Omron CX-Programmer project NewProject (CX-Programmer 9.75)

# PLC PLCGROUP4: CPM2* 

## Global symbols (name address type ; comment)
0.00 BOOL  ; GO_Default
0.01 BOOL  ; IN_PB_1
0.02 BOOL  ; IN_PB_2
0.03 BOOL  ; IN_PB_3
0.04 BOOL  ; SF_FLOOR_1
0.05 BOOL  ; SF_FLOOR_2
0.06 BOOL  ; SF_FLOOR_3
0.07 BOOL  ; SD_CAGE_LIMIT_OPEN
0.08 BOOL  ; SD_CAGE_LIMIT_CLOSE
0.09 BOOL  ; S1_OPEN
0.10 BOOL  ; S1_CLOSE
0.11 BOOL  ; SF_FLOOR_1
0.12 BOOL  ; SF_FLOOR_2
0.13 BOOL  ; SF_FLOOR_3
0.14 BOOL  ; CD_CAGE_LIMIT_OPEN
0.15 BOOL  ; SD_CAGE_LIMIT_CLOSE
10.00 BOOL  ; MOTOR_UP
10.01 BOOL  ; MOTOR_DOWN
10.02 BOOL  ; OPEN_CABIN
10.03 BOOL  ; CLOSE_CABIN
10.04 BOOL  ; M1_OPEN
10.05 BOOL  ; M1_CLOSE
10.06 BOOL  ; M2_OPEN
10.07 BOOL  ; M2_CLOSE
11.00 BOOL  ; M3_OPEN
11.01 BOOL  ; M3_CLOSE
1.00 BOOL  ; S2_OPEN
1.01 BOOL  ; S2_CLOSED
1.02 BOOL  ; S3_OPEN
1.03 BOOL  ; S3_CLOSED
1.04 BOOL  ; SD_CAGE_LIMIT_OPEN
1.05 BOOL  ; SD_CAGE_LIMIT_CLOSE
9.00 BOOL  ; GO_FLOOR_1
9.01 BOOL  ; GO_FLOOR_2
9.02 BOOL  ; GO_FLOOR_3
9.03 BOOL  ; GO_DOWN_FLAG
9.04 BOOL  ; GO_UP_FLAG
9.05 BOOL  ; OPEN_CABIN/FLOOR_DOOR
9.06 BOOL  ; OPEN_DOOR_F1
9.07 BOOL  ; OPEN_DOOR_F2
9.08 BOOL  ; OPEN_DOOR_F3
9.09 BOOL  ; DONE_1
9.10 BOOL  ; DONE_2
9.11 BOOL  ; DONE_3
TIM000 BOOL  ; TIMER CABIN
TIM001 BOOL  ; TIMER_FLOOR_1_DOOR
TIM002 BOOL  ; TIMER_FLOOR_2_DOOR
TIM004 BOOL  ; \

## Program NewProgram1 (no task)
; Lift Code
Local symbols
SF_FLOOR_3 BOOL

### Section Test_Code

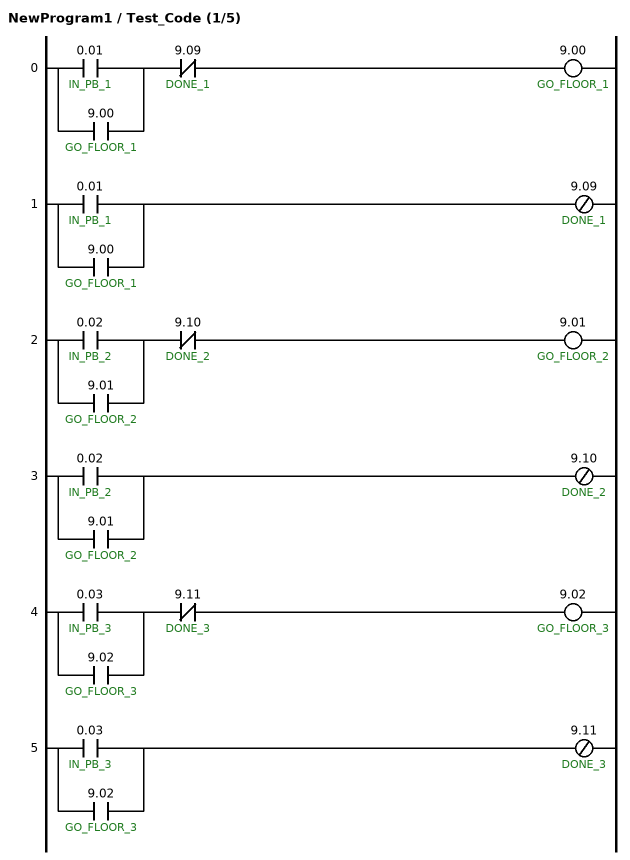
; rung 0
LD 0.01  ; IN_PB_1
OR 9.00  ; GO_FLOOR_1
ANDNOT 9.09  ; DONE_1
OUT 9.00  ; GO_FLOOR_1
; rung 1
LD 0.01  ; IN_PB_1
OR 9.00  ; GO_FLOOR_1
OUTNOT 9.09  ; DONE_1
; rung 2
LD 0.02  ; IN_PB_2
OR 9.01  ; GO_FLOOR_2
ANDNOT 9.10  ; DONE_2
OUT 9.01  ; GO_FLOOR_2
; rung 3
LD 0.02  ; IN_PB_2
OR 9.01  ; GO_FLOOR_2
OUTNOT 9.10  ; DONE_2
; rung 4
LD 0.03  ; IN_PB_3
OR 9.02  ; GO_FLOOR_3
ANDNOT 9.11  ; DONE_3
OUT 9.02  ; GO_FLOOR_3
; rung 5
LD 0.03  ; IN_PB_3
OR 9.02  ; GO_FLOOR_3
OUTNOT 9.11  ; DONE_3

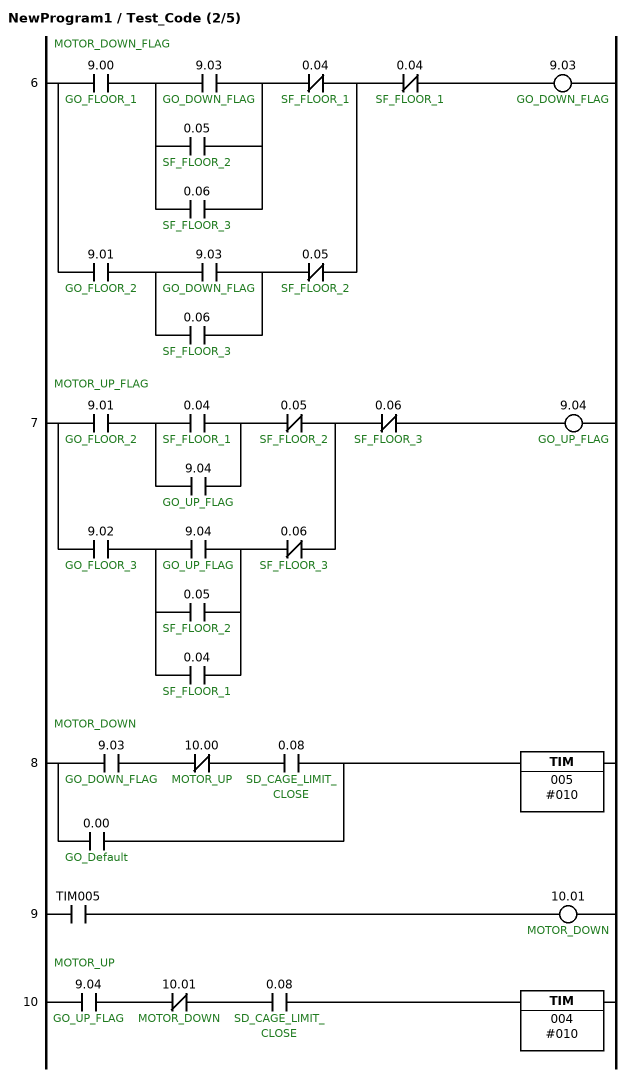
; rung 6: MOTOR_DOWN_FLAG
LD 9.00  ; GO_FLOOR_1
LD 9.03  ; GO_DOWN_FLAG
OR 0.05  ; SF_FLOOR_2
OR 0.06  ; SF_FLOOR_3
ANDLD
ANDNOT 0.04  ; SF_FLOOR_1
LD 9.01  ; GO_FLOOR_2
LD 9.03  ; GO_DOWN_FLAG
OR 0.06  ; SF_FLOOR_3
ANDLD
ANDNOT 0.05  ; SF_FLOOR_2
ORLD
ANDNOT 0.04  ; SF_FLOOR_1
OUT 9.03  ; GO_DOWN_FLAG
; rung 7: MOTOR_UP_FLAG
LD 9.01  ; GO_FLOOR_2
LD 0.04  ; SF_FLOOR_1
OR 9.04  ; GO_UP_FLAG
ANDLD
ANDNOT 0.05  ; SF_FLOOR_2
LD 9.02  ; GO_FLOOR_3
LD 9.04  ; GO_UP_FLAG
OR 0.05  ; SF_FLOOR_2
OR 0.04  ; SF_FLOOR_1
ANDLD
ANDNOT 0.06  ; SF_FLOOR_3
ORLD
ANDNOT 0.06  ; SF_FLOOR_3
OUT 9.04  ; GO_UP_FLAG
; rung 8: MOTOR_DOWN
LD 9.03  ; GO_DOWN_FLAG
ANDNOT 10.00  ; MOTOR_UP
AND 0.08  ; SD_CAGE_LIMIT_CLOSE
OR 0.00  ; GO_Default
TIM 005 #010
; rung 9
LD TIM005
OUT 10.01  ; MOTOR_DOWN
; rung 10: MOTOR_UP
LD 9.04  ; GO_UP_FLAG
ANDNOT 10.01  ; MOTOR_DOWN
AND 0.08  ; SD_CAGE_LIMIT_CLOSE
TIM 004 #010

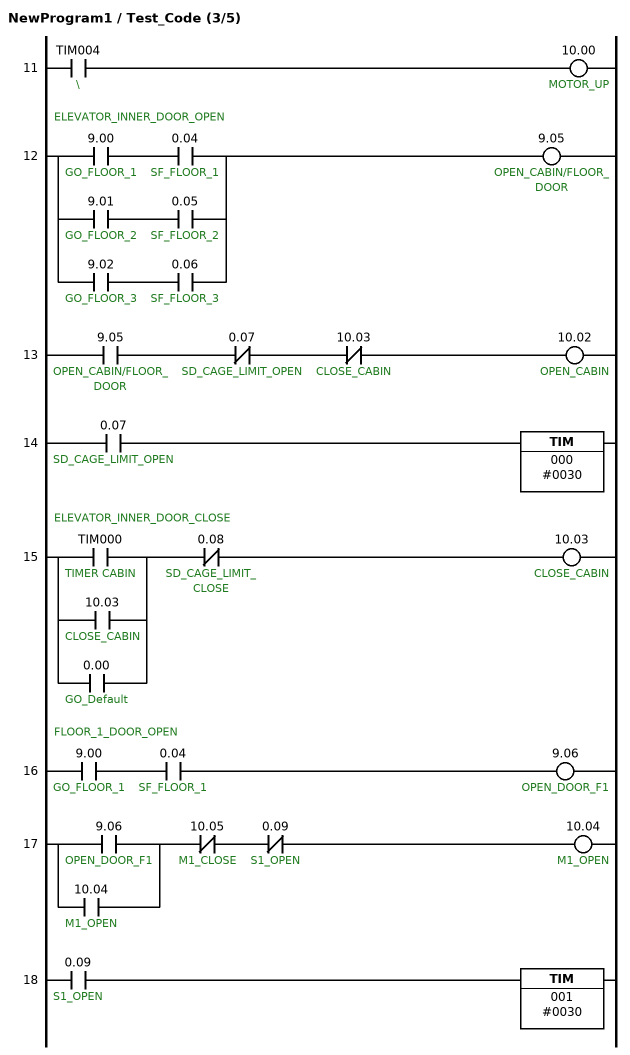
; rung 11
LD TIM004  ; \
OUT 10.00  ; MOTOR_UP
; rung 12: ELEVATOR_INNER_DOOR_OPEN
LD 9.00  ; GO_FLOOR_1
AND 0.04  ; SF_FLOOR_1
LD 9.01  ; GO_FLOOR_2
AND 0.05  ; SF_FLOOR_2
ORLD
LD 9.02  ; GO_FLOOR_3
AND 0.06  ; SF_FLOOR_3
ORLD
OUT 9.05  ; OPEN_CABIN/FLOOR_DOOR
; rung 13
LD 9.05  ; OPEN_CABIN/FLOOR_DOOR
ANDNOT 0.07  ; SD_CAGE_LIMIT_OPEN
ANDNOT 10.03  ; CLOSE_CABIN
OUT 10.02  ; OPEN_CABIN
; rung 14
LD 0.07  ; SD_CAGE_LIMIT_OPEN
TIM 000 #0030
; rung 15: ELEVATOR_INNER_DOOR_CLOSE
LD TIM000  ; TIMER CABIN
OR 10.03  ; CLOSE_CABIN
OR 0.00  ; GO_Default
ANDNOT 0.08  ; SD_CAGE_LIMIT_CLOSE
OUT 10.03  ; CLOSE_CABIN
; rung 16: FLOOR_1_DOOR_OPEN
LD 9.00  ; GO_FLOOR_1
AND 0.04  ; SF_FLOOR_1
OUT 9.06  ; OPEN_DOOR_F1
; rung 17
LD 9.06  ; OPEN_DOOR_F1
OR 10.04  ; M1_OPEN
ANDNOT 10.05  ; M1_CLOSE
ANDNOT 0.09  ; S1_OPEN
OUT 10.04  ; M1_OPEN
; rung 18
LD 0.09  ; S1_OPEN
TIM 001 #0030

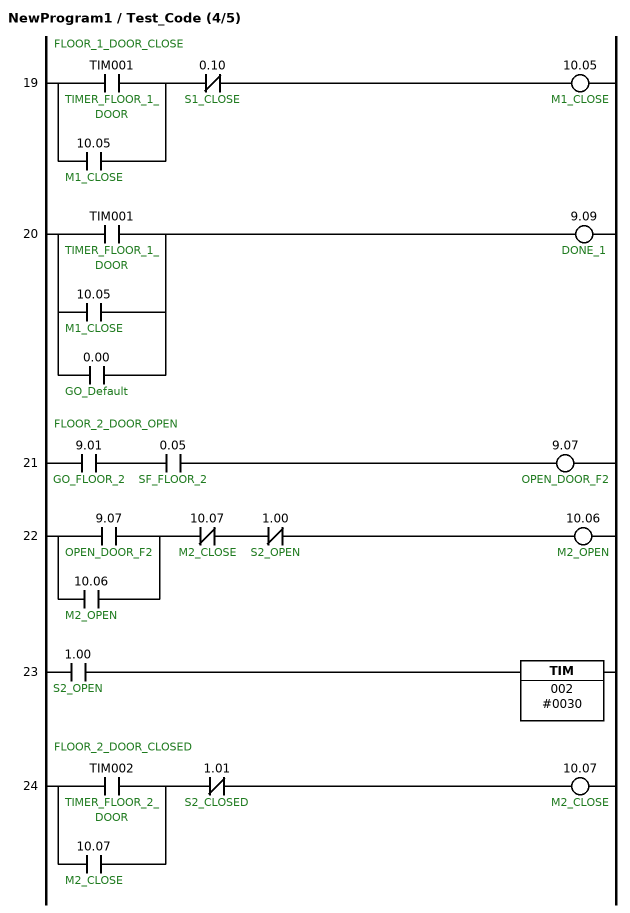
; rung 19: FLOOR_1_DOOR_CLOSE
LD TIM001  ; TIMER_FLOOR_1_DOOR
OR 10.05  ; M1_CLOSE
ANDNOT 0.10  ; S1_CLOSE
OUT 10.05  ; M1_CLOSE
; rung 20
LD TIM001  ; TIMER_FLOOR_1_DOOR
OR 10.05  ; M1_CLOSE
OR 0.00  ; GO_Default
OUT 9.09  ; DONE_1
; rung 21: FLOOR_2_DOOR_OPEN
LD 9.01  ; GO_FLOOR_2
AND 0.05  ; SF_FLOOR_2
OUT 9.07  ; OPEN_DOOR_F2
; rung 22
LD 9.07  ; OPEN_DOOR_F2
OR 10.06  ; M2_OPEN
ANDNOT 10.07  ; M2_CLOSE
ANDNOT 1.00  ; S2_OPEN
OUT 10.06  ; M2_OPEN
; rung 23
LD 1.00  ; S2_OPEN
TIM 002 #0030
; rung 24: FLOOR_2_DOOR_CLOSED
LD TIM002  ; TIMER_FLOOR_2_DOOR
OR 10.07  ; M2_CLOSE
ANDNOT 1.01  ; S2_CLOSED
OUT 10.07  ; M2_CLOSE

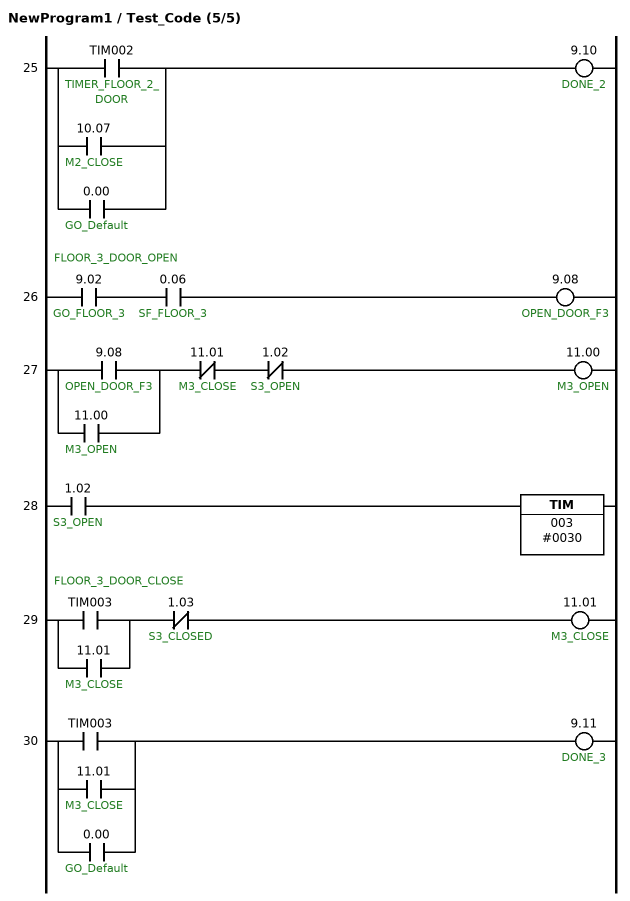
; rung 25
LD TIM002  ; TIMER_FLOOR_2_DOOR
OR 10.07  ; M2_CLOSE
OR 0.00  ; GO_Default
OUT 9.10  ; DONE_2
; rung 26: FLOOR_3_DOOR_OPEN
LD 9.02  ; GO_FLOOR_3
AND 0.06  ; SF_FLOOR_3
OUT 9.08  ; OPEN_DOOR_F3
; rung 27
LD 9.08  ; OPEN_DOOR_F3
OR 11.00  ; M3_OPEN
ANDNOT 11.01  ; M3_CLOSE
ANDNOT 1.02  ; S3_OPEN
OUT 11.00  ; M3_OPEN
; rung 28
LD 1.02  ; S3_OPEN
TIM 003 #0030
; rung 29: FLOOR_3_DOOR_CLOSE
LD TIM003
OR 11.01  ; M3_CLOSE
ANDNOT 1.03  ; S3_CLOSED
OUT 11.01  ; M3_CLOSE
; rung 30
LD TIM003
OR 11.01  ; M3_CLOSE
OR 0.00  ; GO_Default
OUT 9.11  ; DONE_3

### Section END
; rung 0
END(01)